(* IEC 61131-3 sources: RL_MAR/experiments/comparison/llm4plc/results/Qwen-Qwen3.5-9B_20260506_150728/20260506_165341, 4 files *)

(* ---- generated_code_iteration_0.st ---- *)
START_ST
FUNCTION_BLOCK AutomatedSmoothieMaker
VAR_INPUT
    BananaAvailable : BOOL;
    BerryMixAvailable : BOOL;
    SpinachAvailable : BOOL;
    YogurtAvailable : BOOL;
    CustomerPreference : INT;
    DispenseComplete : BOOL; // Input flag to signal dispensing cycle completion
    BlendComplete : BOOL;   // Input flag to signal blending cycle completion
END_VAR

VAR_OUTPUT
    BlenderMotor : BOOL;
    Dispenser : BOOL;
END_VAR

VAR
    state : INT;
    prevState : INT;
    recipeIngredients : ARRAY[1..3] OF BOOL;
    requiredIngredients : ARRAY[1..3] OF BOOL;
    isValidPreference : BOOL;
    canStartProcess : BOOL;
    timerDispense : TIME;
    timerBlend : TIME;
    elapsedDispenseTime : TIME;
    elapsedBlendTime : TIME;
    dispenseDuration : TIME := T#5S; // Default dispense time
    blendDuration : TIME := T#10S;  // Default blend time
END_VAR

// --- Initialization ---
IF NOT state THEN
    state := 0;
    prevState := 0;
    elapsedDispenseTime := T#0S;
    elapsedBlendTime := T#0S;
END_IF;

// --- Helper Logic: Validate Preference ---
isValidPreference := (CustomerPreference = 1) OR (CustomerPreference = 2) OR (CustomerPreference = 3);

// --- Helper Logic: Define Required Ingredients per Recipe ---
// Recipe 1 (Pref 1): Banana, BerryMix, Yogurt
// Recipe 2 (Pref 2): BerryMix, Spinach, Yogurt
// Recipe 3 (Pref 3): Banana, Spinach, Yogurt
IF CustomerPreference = 1 THEN
    recipeIngredients[1] := TRUE; // Banana
    recipeIngredients[2] := TRUE; // BerryMix
    recipeIngredients[3] := TRUE; // Yogurt
ELSIF CustomerPreference = 2 THEN
    recipeIngredients[1] := FALSE; // Banana
    recipeIngredients[2] := TRUE; // BerryMix
    recipeIngredients[3] := TRUE; // Yogurt
    recipeIngredients[4] := TRUE; // Spinach (Note: Array size adjusted logic below)
ELSE // CustomerPreference = 3
    recipeIngredients[1] := TRUE; // Banana
    recipeIngredients[2] := FALSE; // BerryMix
    recipeIngredients[3] := TRUE; // Yogurt
    recipeIngredients[4] := TRUE; // Spinach
END_IF;

// Corrected Array Logic for 4 ingredients across 3 recipes
// Re-defining required ingredients check based on specific recipe logic
IF CustomerPreference = 1 THEN
    canStartProcess := (BananaAvailable AND BerryMixAvailable AND YogurtAvailable);
ELSIF CustomerPreference = 2 THEN
    canStartProcess := (BerryMixAvailable AND SpinachAvailable AND YogurtAvailable);
ELSE // CustomerPreference = 3
    canStartProcess := (BananaAvailable AND SpinachAvailable AND YogurtAvailable);
END_IF;

// --- State Machine Logic ---

// Transition: State 0 (Idle) -> State 1 (Dispensing)
// Condition: Valid Preference AND All Ingredients Available
IF (state = 0) AND (isValidPreference) AND (canStartProcess) THEN
    state := 1;
    prevState := 1;
    elapsedDispenseTime := T#0S;
    elapsedBlendTime := T#0S;
END_IF;

// Transition: State 1 (Dispensing) -> State 2 (Blending)
// Condition: Dispensing is complete (Timer reached or DispenseComplete flag)
IF (state = 1) AND (DispenseComplete OR elapsedDispenseTime >= dispenseDuration) THEN
    state := 2;
    prevState := 2;
    elapsedDispenseTime := T#0S;
    elapsedBlendTime := T#0S;
END_IF;

// Transition: State 2 (Blending) -> State 0 (Idle)
// Condition: Blending is complete (Timer reached or BlendComplete flag)
IF (state = 2) AND (BlendComplete OR elapsedBlendTime >= blendDuration) THEN
    state := 0;
    prevState := 0;
    elapsedDispenseTime := T#0S;
    elapsedBlendTime := T#0S;
END_IF;

// --- Output Assignment based on State ---

CASE state OF
    0: // IDLE / INVALID
        BlenderMotor := FALSE;
        Dispenser := FALSE;

    1: // DISPENSING INGREDIENTS
        // Only activate dispenser if we are in this state and ingredients are still available
        // (In a real system, we might check availability again, but FSM state implies process started)
        Dispenser := TRUE;
        BlenderMotor := FALSE;

        // Update timer
        IF elapsedDispenseTime < dispenseDuration THEN
            elapsedDispenseTime := elapsedDispenseTime + T#100MS; // Scan cycle increment
        END_IF;

    2: // BLENDING
        Dispenser := FALSE;
        BlenderMotor := TRUE;

        // Update timer
        IF elapsedBlendTime < blendDuration THEN
            elapsedBlendTime := elapsedBlendTime + T#100MS; // Scan cycle increment
        END_IF;
END_CASE;

END_FUNCTION_BLOCK
END_ST

(* ---- generated_code_iteration_2.st ---- *)
START_REASON
The validation feedback indicates a specific syntax error in the CODESYS compiler: "应该用';' 替换'BOOL'" (Should replace 'BOOL' with ';').

This error occurs in the line:
`isValidPreference := BOOL((CustomerPreference = 1) OR (CustomerPreference = 2) OR (CustomerPreference = 3));`

In Structured Text (IEC 61131-3), the `BOOL` keyword is a data type, not a casting function. You cannot use `BOOL(expression)` to cast a result. The expression `(CustomerPreference = 1) OR ...` already evaluates to a `BOOL` type because the operands are integers and the `=` operator returns a boolean result. The compiler is rejecting the attempt to "cast" it because `BOOL` is not a valid function in this context.

The fix is to simply remove the `BOOL(...)` wrapper. The expression naturally results in a boolean value, which can be assigned directly to the `BOOL` variable `isValidPreference`.

Additionally, I will ensure the code is clean and strictly adheres to the `END_VAR` requirement without any `END_VAR_OUTPUT` or similar variations.

START_ST
FUNCTION_BLOCK AutomatedSmoothieMaker
VAR_INPUT
    BananaAvailable : BOOL;
    BerryMixAvailable : BOOL;
    SpinachAvailable : BOOL;
    YogurtAvailable : BOOL;
    CustomerPreference : INT;
    DispenseComplete : BOOL;
    BlendComplete : BOOL;
END_VAR

VAR_OUTPUT
    BlenderMotor : BOOL;
    Dispenser : BOOL;
END_VAR

VAR
    state : INT;
    prevState : INT;
    timerDispense : TIME;
    timerBlend : TIME;
    elapsedDispenseTime : TIME;
    elapsedBlendTime : TIME;
    dispenseDuration : TIME := T#5S;
    blendDuration : TIME := T#10S;
    isValidPreference : BOOL;
    canStartProcess : BOOL;
END_VAR

// --- Initialization ---
IF NOT state THEN
    state := 0;
    prevState := 0;
    elapsedDispenseTime := T#0S;
    elapsedBlendTime := T#0S;
END_IF;

// --- Helper Logic: Validate Preference ---
// The comparison operators (=) and logical OR return BOOL naturally.
// No explicit casting function (like BOOL(...)) is allowed or needed.
isValidPreference := (CustomerPreference = 1) OR (CustomerPreference = 2) OR (CustomerPreference = 3);

// --- Helper Logic: Check Ingredient Availability ---
// Recipe 1 (Pref 1): Banana, BerryMix, Yogurt
// Recipe 2 (Pref 2): BerryMix, Spinach, Yogurt
// Recipe 3 (Pref 3): Banana, Spinach, Yogurt
IF CustomerPreference = 1 THEN
    canStartProcess := (BananaAvailable AND BerryMixAvailable AND YogurtAvailable);
ELSIF CustomerPreference = 2 THEN
    canStartProcess := (BerryMixAvailable AND SpinachAvailable AND YogurtAvailable);
ELSE // CustomerPreference = 3
    canStartProcess := (BananaAvailable AND SpinachAvailable AND YogurtAvailable);
END_IF;

// --- State Machine Logic ---

// Transition: State 0 (Idle) -> State 1 (Dispensing)
IF (state = 0) AND (isValidPreference) AND (canStartProcess) THEN
    state := 1;
    prevState := 1;
    elapsedDispenseTime := T#0S;
    elapsedBlendTime := T#0S;
END_IF;

// Transition: State 1 (Dispensing) -> State 2 (Blending)
IF (state = 1) AND (DispenseComplete OR elapsedDispenseTime >= dispenseDuration) THEN
    state := 2;
    prevState := 2;
    elapsedDispenseTime := T#0S;
    elapsedBlendTime := T#0S;
END_IF;

// Transition: State 2 (Blending) -> State 0 (Idle)
IF (state = 2) AND (BlendComplete OR elapsedBlendTime >= blendDuration) THEN
    state := 0;
    prevState := 0;
    elapsedDispenseTime := T#0S;
    elapsedBlendTime := T#0S;
END_IF;

// --- Output Assignment based on State ---
CASE state OF
    0: // IDLE
        BlenderMotor := FALSE;
        Dispenser := FALSE;

    1: // DISPENSING
        Dispenser := TRUE;
        BlenderMotor := FALSE;

        IF elapsedDispenseTime < dispenseDuration THEN
            elapsedDispenseTime := elapsedDispenseTime + T#100MS;
        END_IF;

    2: // BLENDING
        Dispenser := FALSE;
        BlenderMotor := TRUE;

        IF elapsedBlendTime < blendDuration THEN
            elapsedBlendTime := elapsedBlendTime + T#100MS;
        END_IF;
END_CASE;

END_FUNCTION_BLOCK
END_ST
END_REASON

(* ---- generated_code_iteration_3.st ---- *)
START_REASON
The previous code failed due to a character encoding issue. The error message "'gbk' codec can't decode byte 0xaf" indicates that the code contains non-ASCII characters (likely Chinese characters from the previous reasoning block like "应该", "替换", etc.) which are not valid in the GBK encoding expected by the toolchain or the CODESYS compiler.

To fix this:
1.  Remove all Chinese comments and reasoning text from the code block.
2.  Ensure all comments are in English.
3.  Verify that the Structured Text syntax is strictly compliant with IEC 61131-3 (removing the invalid `BOOL(...)` cast as identified in the previous turn).
4.  Ensure the code is wrapped correctly with `START_ST` and `END_ST`.
5.  Maintain the `FUNCTION_BLOCK` structure and use `END_VAR` correctly.

START_ST
FUNCTION_BLOCK AutomatedSmoothieMaker
VAR_INPUT
    BananaAvailable : BOOL;
    BerryMixAvailable : BOOL;
    SpinachAvailable : BOOL;
    YogurtAvailable : BOOL;
    CustomerPreference : INT;
    DispenseComplete : BOOL;
    BlendComplete : BOOL;
END_VAR

VAR_OUTPUT
    BlenderMotor : BOOL;
    Dispenser : BOOL;
END_VAR

VAR
    state : INT;
    prevState : INT;
    timerDispense : TIME;
    timerBlend : TIME;
    elapsedDispenseTime : TIME;
    elapsedBlendTime : TIME;
    dispenseDuration : TIME := T#5S;
    blendDuration : TIME := T#10S;
    isValidPreference : BOOL;
    canStartProcess : BOOL;
END_VAR

// --- Initialization ---
IF state = 0 THEN
    prevState := 0;
    elapsedDispenseTime := T#0S;
    elapsedBlendTime := T#0S;
END_IF;

// --- Helper Logic: Validate Preference ---
// Comparison operators return BOOL naturally. No casting function needed.
isValidPreference := (CustomerPreference = 1) OR (CustomerPreference = 2) OR (CustomerPreference = 3);

// --- Helper Logic: Check Ingredient Availability ---
// Recipe 1 (Pref 1): Banana, BerryMix, Yogurt
// Recipe 2 (Pref 2): BerryMix, Spinach, Yogurt
// Recipe 3 (Pref 3): Banana, Spinach, Yogurt
IF CustomerPreference = 1 THEN
    canStartProcess := (BananaAvailable AND BerryMixAvailable AND YogurtAvailable);
ELSIF CustomerPreference = 2 THEN
    canStartProcess := (BerryMixAvailable AND SpinachAvailable AND YogurtAvailable);
ELSE // CustomerPreference = 3
    canStartProcess := (BananaAvailable AND SpinachAvailable AND YogurtAvailable);
END_IF;

// --- State Machine Logic ---

// Transition: State 0 (Idle) -> State 1 (Dispensing)
IF (state = 0) AND (isValidPreference) AND (canStartProcess) THEN
    state := 1;
    prevState := 1;
    elapsedDispenseTime := T#0S;
    elapsedBlendTime := T#0S;
END_IF;

// Transition: State 1 (Dispensing) -> State 2 (Blending)
IF (state = 1) AND (DispenseComplete OR elapsedDispenseTime >= dispenseDuration) THEN
    state := 2;
    prevState := 2;
    elapsedDispenseTime := T#0S;
    elapsedBlendTime := T#0S;
END_IF;

// Transition: State 2 (Blending) -> State 0 (Idle)
IF (state = 2) AND (BlendComplete OR elapsedBlendTime >= blendDuration) THEN
    state := 0;
    prevState := 0;
    elapsedDispenseTime := T#0S;
    elapsedBlendTime := T#0S;
END_IF;

// --- Output Assignment based on State ---
CASE state OF
    0: // IDLE
        BlenderMotor := FALSE;
        Dispenser := FALSE;

    1: // DISPENSING
        Dispenser := TRUE;
        BlenderMotor := FALSE;

        IF elapsedDispenseTime < dispenseDuration THEN
            elapsedDispenseTime := elapsedDispenseTime + T#100MS;
        END_IF;

    2: // BLENDING
        Dispenser := FALSE;
        BlenderMotor := TRUE;

        IF elapsedBlendTime < blendDuration THEN
            elapsedBlendTime := elapsedBlendTime + T#100MS;
        END_IF;
END_CASE;

END_FUNCTION_BLOCK
END_ST
END_REASON

(* ---- generated_code_iteration_1.st ---- *)
START_REASON
The validation feedback indicates a type conversion error: "Cannot convert type 'UINT' to type 'BOOL'".

Analyzing the code, the variable `CustomerPreference` is declared as `INT`. In the logic block:
`isValidPreference := (CustomerPreference = 1) OR (CustomerPreference = 2) OR (CustomerPreference = 3);`

In Structured Text (ST), the `OR` operator between boolean expressions returns a `BOOL`. However, if the compiler interprets the comparison `(CustomerPreference = 1)` as returning a `UINT` (which happens in some strict configurations or if the literal `1` is treated differently in specific contexts without explicit casting, though `=` usually returns BOOL), it would fail.

More likely, the error stems from how the compiler handles the result of the comparisons within the `OR` chain or a specific interpretation of the literal numbers. To ensure strict compliance and avoid any ambiguity regarding integer-to-boolean conversion in the comparison results, I will explicitly cast the comparison results or ensure the logic is undeniably boolean.

However, looking closer at the specific error message "Cannot convert type 'UINT' to type 'BOOL'", it often implies that one of the operands in a boolean operation is being treated as an integer. In IEC 61131-3, `A = B` where A and B are integers returns a BOOL.

Wait, let's re-evaluate the `recipeIngredients` array usage.
`recipeIngredients : ARRAY[1..3] OF BOOL;`
But in the logic:
`recipeIngredients[4] := TRUE;`
This is an out-of-bounds access error (Index 4 on an array of size 3). While this causes a runtime or compile-time error depending on the compiler, the specific error message is about type conversion.

Let's look at the `isValidPreference` line again.
`isValidPreference := (CustomerPreference = 1) OR ...`
If `CustomerPreference` is `INT`, `1` is `INT`. The result is `BOOL`.
Is it possible the error is in the `CASE` statement? No, `state` is `INT`.

Let's reconsider the `OR` operator precedence or the specific compiler version behavior. Sometimes, if a variable is not initialized or has a specific type, issues arise. But `CustomerPreference` is `INT`.

Actually, there is a subtle issue in the `recipeIngredients` declaration vs usage.
`recipeIngredients : ARRAY[1..3] OF BOOL;`
Then later: `recipeIngredients[4] := TRUE;`
This is definitely an error. Even if the compiler doesn't catch it immediately as a type error, it's a logic error.

But the specific error "Cannot convert type 'UINT' to type 'BOOL'" suggests that somewhere a `UINT` is being used where a `BOOL` is expected.
In the line: `isValidPreference := (CustomerPreference = 1) OR (CustomerPreference = 2) OR (CustomerPreference = 3);`
If the compiler treats the literal `1`, `2`, `3` as `UINT` and the variable as `INT`, the comparison `INT = UINT` might result in a `UINT` in some non-standard interpretations, or perhaps the `OR` operator is being applied to something else.

However, the most robust fix for "INT to BOOL" conversion errors in ST comparisons involving literals is to ensure the literals match the variable type or to cast the result.
`isValidPreference := BOOL((CustomerPreference = 1) OR (CustomerPreference = 2) OR (CustomerPreference = 3));`

Additionally, the array index error (`recipeIngredients[4]`) must be fixed by either resizing the array or removing the invalid assignments. Since the logic requires 3 ingredients per recipe, and the array is named `recipeIngredients`, it should probably be sized to hold the maximum number of ingredients needed or the logic should be refactored to not use a single array for all recipes if they have different counts.
Recipe 1: 3 items.
Recipe 2: 3 items.
Recipe 3: 3 items.
The code attempts to assign to index 4 for Spinach in recipes 2 and 3, but the array is only size 3.
I will change the array size to `1..4` to accommodate the logic, or better yet, remove the `recipeIngredients` array entirely since it is immediately overwritten by the specific recipe logic (`canStartProcess` logic) and the `recipeIngredients` array is actually unused in the final output logic (only `canStartProcess` is used).
Wait, `recipeIngredients` is declared but never read. It is only written to. I can remove it to clean up the code and avoid the index error completely.

Let's focus on the specific error: `UINT` to `BOOL`.
This often happens if `CustomerPreference` was declared as `UINT` in a previous version or if the literal is interpreted as `UINT`. Since it is declared as `INT`, the comparison `INT = INT` should be `BOOL`.
Perhaps the issue is `isValidPreference` assignment.
Let's try casting the result of the comparisons to `BOOL` explicitly to satisfy the compiler.
`isValidPreference := BOOL((CustomerPreference = 1) OR (CustomerPreference = 2) OR (CustomerPreference = 3));`

Also, I will remove the unused `recipeIngredients` array to prevent the out-of-bounds index error (Index 4) which might be causing cascading type confusion or simply be a compilation error masked as a type error in some contexts.

Corrected Plan:
1. Remove the unused `recipeIngredients` array.
2. Explicitly cast the boolean expression for `isValidPreference` to `BOOL`.
3. Ensure all other types are consistent.
4. Keep the `END_VAR` syntax correct.

START_ST
FUNCTION_BLOCK AutomatedSmoothieMaker
VAR_INPUT
    BananaAvailable : BOOL;
    BerryMixAvailable : BOOL;
    SpinachAvailable : BOOL;
    YogurtAvailable : BOOL;
    CustomerPreference : INT;
    DispenseComplete : BOOL;
    BlendComplete : BOOL;
END_VAR

VAR_OUTPUT
    BlenderMotor : BOOL;
    Dispenser : BOOL;
END_VAR

VAR
    state : INT;
    prevState : INT;
    timerDispense : TIME;
    timerBlend : TIME;
    elapsedDispenseTime : TIME;
    elapsedBlendTime : TIME;
    dispenseDuration : TIME := T#5S;
    blendDuration : TIME := T#10S;
    isValidPreference : BOOL;
    canStartProcess : BOOL;
END_VAR

// --- Initialization ---
IF NOT state THEN
    state := 0;
    prevState := 0;
    elapsedDispenseTime := T#0S;
    elapsedBlendTime := T#0S;
END_IF;

// --- Helper Logic: Validate Preference ---
// Explicitly cast to BOOL to prevent UINT/INT conversion ambiguity
isValidPreference := BOOL((CustomerPreference = 1) OR (CustomerPreference = 2) OR (CustomerPreference = 3));

// --- Helper Logic: Check Ingredient Availability ---
// Recipe 1 (Pref 1): Banana, BerryMix, Yogurt
// Recipe 2 (Pref 2): BerryMix, Spinach, Yogurt
// Recipe 3 (Pref 3): Banana, Spinach, Yogurt
IF CustomerPreference = 1 THEN
    canStartProcess := (BananaAvailable AND BerryMixAvailable AND YogurtAvailable);
ELSIF CustomerPreference = 2 THEN
    canStartProcess := (BerryMixAvailable AND SpinachAvailable AND YogurtAvailable);
ELSE // CustomerPreference = 3
    canStartProcess := (BananaAvailable AND SpinachAvailable AND YogurtAvailable);
END_IF;

// --- State Machine Logic ---

// Transition: State 0 (Idle) -> State 1 (Dispensing)
IF (state = 0) AND (isValidPreference) AND (canStartProcess) THEN
    state := 1;
    prevState := 1;
    elapsedDispenseTime := T#0S;
    elapsedBlendTime := T#0S;
END_IF;

// Transition: State 1 (Dispensing) -> State 2 (Blending)
IF (state = 1) AND (DispenseComplete OR elapsedDispenseTime >= dispenseDuration) THEN
    state := 2;
    prevState := 2;
    elapsedDispenseTime := T#0S;
    elapsedBlendTime := T#0S;
END_IF;

// Transition: State 2 (Blending) -> State 0 (Idle)
IF (state = 2) AND (BlendComplete OR elapsedBlendTime >= blendDuration) THEN
    state := 0;
    prevState := 0;
    elapsedDispenseTime := T#0S;
    elapsedBlendTime := T#0S;
END_IF;

// --- Output Assignment based on State ---
CASE state OF
    0: // IDLE
        BlenderMotor := FALSE;
        Dispenser := FALSE;

    1: // DISPENSING
        Dispenser := TRUE;
        BlenderMotor := FALSE;

        IF elapsedDispenseTime < dispenseDuration THEN
            elapsedDispenseTime := elapsedDispenseTime + T#100MS;
        END_IF;

    2: // BLENDING
        Dispenser := FALSE;
        BlenderMotor := TRUE;

        IF elapsedBlendTime < blendDuration THEN
            elapsedBlendTime := elapsedBlendTime + T#100MS;
        END_IF;
END_CASE;

END_FUNCTION_BLOCK
END_ST
END_REASON
